// TwinCAT 3 PLC project PLC01
// ProgramVersion: 3.1.4024.0
// libraries:
//   Tc2_EtherCAT, * (Beckhoff Automation GmbH)
//   Tc2_Standard, * (Beckhoff Automation GmbH)
//   Tc2_System, * (Beckhoff Automation GmbH)
//   Tc2_Utilities, * (Beckhoff Automation GmbH)
//   Tc3_Module, * (Beckhoff Automation GmbH)
// project tree:
//   / GlobalTextList.TcGTLO, PlcTask.TcTTO, Visualization Manager.TcVMO (not stored)
//   GVLs/ G_Safety.TcGVL
//   POUs/ FB_Sample.TcPOU, FB_Teste.TcPOU, MAIN.TcPOU, safetyDiag.TcPOU
//   POUs/SafetyDiag/DUTs/ E_connInfoDiag.TcDUT, st_ConnectionInfoData.TcDUT, st_diagFBBits.TcDUT, st_infoDataFB.TcDUT, st_InfoDataGroup.TcDUT
//   POUs/SafetyDiag/ FB_ConnDiagELx904.TcPOU, FB_ConnectionDiag.TcPOU, FB_EStopDiag.TcPOU, FB_GroupDiag.TcPOU
//   POUs/SafetyDiag/ITF/ I_FBDiag.TcIO
//   VISUs/ ConnDiag.TcVIS, FB_Diag.TcVIS, footer.TcVIS, Group.TcVIS, Visualization.TcVIS
//   VISUs/Frames/ DiagConnELx904.TcVIS, DiagEStop.TcVIS
// real-time tasks:
//   TASK PlcTask: cycle T#10ms, priority 20, ADS port 350
// motion (NC):
//   TASK NC-Task 1 SAF: cycle T#2ms, priority 4, ADS port 501
//   TASK NC-Task 1 SVB: cycle T#10ms, priority 8, ADS port 511
//   AXIS Axis 1 (id 1)
//     OtherSettings: AllowMotionCmdToSlave=true
//     encoder EncType=19
//       EncPara: MaxCount=#xffffffff
//     drive DrvType=16
//       DrvPara: MaxCount=#xffffffff, DriveControlDWord=#x00020000
//         Analog: TorqueSetpointScale=10, ScaleFactorActTorque=0.1
//         TimeComp: TaskDelayCycles=1
//     controller CtrType=1
//       CtrPara: PriorControlFactor=1
//         Observer: BandWidth=20
//   AXIS Axis 2 (id 2)
//     OtherSettings: AllowMotionCmdToSlave=true
//     encoder EncType=19
//       EncPara: MaxCount=#xffffffff
//     drive DrvType=16
//       DrvPara: MaxCount=#xffffffff, DriveControlDWord=#x00020000
//         Analog: TorqueSetpointScale=10, ScaleFactorActTorque=0.1
//         TimeComp: TaskDelayCycles=1
//     controller CtrType=1
//       CtrPara: PriorControlFactor=1
//         Observer: BandWidth=20
// I/O:
//   DEVICE Device 2 (EtherCAT), AmsNetId 192.168.10.7.3.1
//     Term 1 (EK1100) [EK1100 EtherCAT Coupler (2A E-Bus)]
//       Term 2 (EL1012) [EL1012 2Ch. Dig. Input 24V, 10µs]
//       Term 3 (EL1012) [EL1012 2Ch. Dig. Input 24V, 10µs]
//       Term 4 (EL1012) [EL1012 2Ch. Dig. Input 24V, 10µs]
//       Term 5 (EL1012) [EL1012 2Ch. Dig. Input 24V, 10µs]
//       Term 6 (EL2004) [EL2004 4Ch. Dig. Output 24V, 0.5A]
//       Term 7 (EL4002) [EL4002 2Ch. Ana. Output 0-10V, 12bit]
//       Term 8 (EL9512) [EL9512 Power supply terminal 12V]
//       Term 9 (EL3102) [EL3102 2Ch. Ana. Input +/-10V, Diff.]
//       Term 16 (EL9011) [EL9011 End Terminal]
//     Term 10 (EK1100) [EK1100 EtherCAT Coupler (2A E-Bus)]
//       Term 11 (EL7211-0010) [EL7211-0010 1Ch. MDP742 Servo motor output stage with OCT (50V, 4.5A RMS)]
//       Term 12 (EL7211-0010) [EL7211-0010 1Ch. MDP742 Servo motor output stage with OCT (50V, 4.5A RMS)]
//       Term 13 (EL1904) [EL1904, 4 Ch. Safety Input 24V, TwinSAFE]
//         modules: Module 1 (FSOES)
//       Term 14 (EL2904) [EL2904, 4 Ch. Safety Output 24V, 0.5A, TwinSAFE]
//         modules: Module 1 (FSOES), Module 2 (DO)
//       Term 15 (EL6900) [EL6900, TwinSAFE PLC]
//       Term 17 (EL9011) [EL9011 End Terminal]
// variable links:
//   Device 2 (EtherCAT) <-> Device 2 (EtherCAT)/Term 10 (EK1100)/Term 13 (EL1904)
//     Term 10 (EK1100)/Term 15 (EL6900)/ConnectionInputs/Message_2 TxPDO <-> Module 1 (FSOES)/RxPDO/FSOE
//   Device 2 (EtherCAT) <-> Device 2 (EtherCAT)/Term 10 (EK1100)/Term 14 (EL2904)
//     Term 10 (EK1100)/Term 15 (EL6900)/ConnectionOutputs/Message_3 RxPDO <-> Module 1 (FSOES)/TxPDO/FSOE
//   Device 2 (EtherCAT) <-> Device 2 (EtherCAT)/Term 10 (EK1100)/Term 15 (EL6900)
//     Term 10 (EK1100)/Term 13 (EL1904)/Module 1 (FSOES)/TxPDO/FSOE <-> ConnectionOutputs/Message_2 RxPDO
//     Term 10 (EK1100)/Term 14 (EL2904)/Module 1 (FSOES)/RxPDO/FSOE <-> ConnectionInputs/Message_3 TxPDO
//   NC-Task 1 SAF/Axes/Axis 1 <-> Device 2 (EtherCAT)/Term 10 (EK1100)/Term 11 (EL7211-0010)
//     Drive/Inputs/In/nDcOutputTime <-> InfoData/DcOutputShift
//     Drive/Inputs/In/nState1 <-> DRV Statusword/Statusword
//     Drive/Inputs/In/nState2 <-> DRV Statusword/Statusword @bit 8
//     Drive/Inputs/In/nState4 @bit 1 <-> WcState/InputToggle
//     Drive/Inputs/In/nState4 <-> WcState/WcState
//     Drive/Outputs/Out/nCtrl1 <-> DRV Controlword/Controlword
//     Drive/Outputs/Out/nCtrl2 <-> DRV Controlword/Controlword @bit 8
//     Drive/Outputs/Out/nDataOut2 <-> DRV Target velocity/Target velocity
//     Enc/Inputs/In/nDataIn1 <-> FB Position/Position
//     Enc/Inputs/In/nDcInputTime <-> InfoData/DcInputShift
//     Enc/Inputs/In/nState4 @bit 1 <-> WcState/InputToggle
//     Enc/Inputs/In/nState4 <-> WcState/WcState
//   NC-Task 1 SAF/Axes/Axis 2 <-> Device 2 (EtherCAT)/Term 10 (EK1100)/Term 12 (EL7211-0010)
//     Drive/Inputs/In/nDcOutputTime <-> InfoData/DcOutputShift
//     Drive/Inputs/In/nState1 <-> DRV Statusword/Statusword
//     Drive/Inputs/In/nState2 <-> DRV Statusword/Statusword @bit 8
//     Drive/Inputs/In/nState4 @bit 1 <-> WcState/InputToggle
//     Drive/Inputs/In/nState4 <-> WcState/WcState
//     Drive/Outputs/Out/nCtrl1 <-> DRV Controlword/Controlword
//     Drive/Outputs/Out/nCtrl2 <-> DRV Controlword/Controlword @bit 8
//     Drive/Outputs/Out/nDataOut2 <-> DRV Target velocity/Target velocity
//     Enc/Inputs/In/nDataIn1 <-> FB Position/Position
//     Enc/Inputs/In/nDcInputTime <-> InfoData/DcInputShift
//     Enc/Inputs/In/nState4 @bit 1 <-> WcState/InputToggle
//     Enc/Inputs/In/nState4 <-> WcState/WcState
//   PLC01/PLC01 Instance <-> Device 2 (EtherCAT)/Term 10 (EK1100)/Term 15 (EL6900)
//     PlcTask Inputs/safetyDiag.blocoEStop.fbInfoData/diag <-> Function Block Info Data/TwinSafeGroup1.Network1.FBEstop1 Info Data/Diag
//     PlcTask Inputs/safetyDiag.blocoEStop.fbInfoData/state <-> Function Block Info Data/TwinSafeGroup1.Network1.FBEstop1 Info Data/State
//     PlcTask Inputs/safetyDiag.connDiagEL1904.connInfo/bit{1..4} <-> Connection Info Data/Message_2 Info Data/Input Safe Data InputChannel{1..4}  (4 links)
//     PlcTask Inputs/safetyDiag.connDiagEL1904.connInfo/diag <-> Connection Info Data/Message_2 Info Data/Diag
//     PlcTask Inputs/safetyDiag.connDiagEL2904.connInfo/diag <-> Connection Info Data/Message_3 Info Data/Diag
//     PlcTask Inputs/safetyDiag.connDiagEL1904.connInfo/state <-> Connection Info Data/Message_2 Info Data/State
//     PlcTask Inputs/safetyDiag.connDiagEL2904.connInfo/state <-> Connection Info Data/Message_3 Info Data/State
//     PlcTask Inputs/safetyDiag.connDiagEL2904.connInfo/bit{1..4} <-> Connection Info Data/Message_3 Info Data/Output Safe Data OutputChannel{1..4}  (4 links)
//     PlcTask Inputs/safetyDiag.eStopGroup.groupInfoData <-> TwinSAFE Group Info Data/TwinSafeGroup1 Info Data
//     PlcTask Outputs/G_Safety.resetSafety <-> StandardOutputs/Standard In Var 1
//     PlcTask Outputs/G_Safety.runSafety <-> StandardOutputs/Standard In Var 4

CONFIGURATION PLC01
    RESOURCE PLC ON TwinCAT3
        TASK PlcTask(INTERVAL := T#10ms, PRIORITY := 20);
        PROGRAM MAIN WITH PlcTask : MAIN;
    END_RESOURCE
END_CONFIGURATION

// ---- POUs/SafetyDiag/DUTs/E_connInfoDiag.TcDUT
{attribute 'qualified_only'}
{attribute 'strict'}
TYPE E_connInfoDiag :
(
	invalidCommand,
	unknownCommand,
	invalidConnectionId,
	invalidCRC,
	watchdogTime,
	invalidFSOEAddr,
	invalidData,
	invalidCommParaLen,
	invalidCommPara,
	invalidUserParaLen,
	invalidUserPara,
	FSOEMasterReset,
	moduleErrOnSlave,
	moduleErrEl290x,
	slaveNotStarted,
	FSOESlaveErr,
	FSOESlaveFailsafeActive,
	startup,
	FSOEMasterFailsafeActive
);
END_TYPE

// ---- POUs/SafetyDiag/DUTs/st_ConnectionInfoData.TcDUT
TYPE st_ConnectionInfoData :
STRUCT
	state,diag:USINT;
	bit1,bit2,bit3,bit4:BIT;
END_STRUCT
END_TYPE

// ---- POUs/SafetyDiag/DUTs/st_diagFBBits.TcDUT
TYPE st_diagFBBits :ARRAY[0..15] OF BOOL;
END_TYPE

// ---- POUs/SafetyDiag/DUTs/st_infoDataFB.TcDUT
TYPE st_infoDataFB :
STRUCT
	state:USINT;
	diag:UINT;
END_STRUCT
END_TYPE

// ---- POUs/SafetyDiag/DUTs/st_InfoDataGroup.TcDUT
TYPE st_InfoDataGroup :
STRUCT
	state,diag:USINT;
END_STRUCT
END_TYPE

// ---- GVLs/G_Safety.TcGVL
{attribute 'qualified_only'}
VAR_GLOBAL
	runSafety AT %Q*:BOOL;	//ativação do safety
	resetSafety AT %Q*:BOOL;//reset do safety
END_VAR

// ---- POUs/SafetyDiag/ITF/I_FBDiag.TcIO
INTERFACE I_FBDiag

PROPERTY P_diagBits : st_diagFBBits
GET
END_GET
END_PROPERTY

PROPERTY P_State : STRING(20)
GET
END_GET
END_PROPERTY

END_INTERFACE

// ---- POUs/MAIN.TcPOU
PROGRAM MAIN
VAR
	r1:LREAL:=20;
    fbSample : FB_Sample; 
    sMyPath : STRING; 
	teste:FB_Teste;
	grupo:FB_GroupDiag;
END_VAR

safetyDiag();
fbSample(); 
sMyPath := fbSample.sPath;

END_PROGRAM

// ---- POUs/FB_Sample.TcPOU
{attribute 'reflection'} 
FUNCTION_BLOCK FB_Sample 
VAR 
    {attribute 'instance-path'} 
    {attribute 'noinit'} 
    sPath : STRING; 
END_VAR

END_FUNCTION_BLOCK

// ---- POUs/FB_Teste.TcPOU
{attribute 'reflection'} 
FUNCTION_BLOCK FB_Teste
VAR
    {attribute 'instance-path'} 
    {attribute 'noinit'} 
	varTeste:STRING;
END_VAR

END_FUNCTION_BLOCK

// ---- POUs/SafetyDiag/FB_GroupDiag.TcPOU
{attribute 'reflection'} 
FUNCTION_BLOCK FB_GroupDiag
VAR_INPUT
	logGroupErrorState:BOOL:=TRUE;
END_VAR
VAR
    {attribute 'instance-path'}
    {attribute 'noinit'}
	sPath:STRING;	
	groupInfoData AT %I*:st_InfoDataGroup;
	oldGroupState:USINT;
	sCurrDiag:STRING(20);
END_VAR

PROPERTY diagInfo : string(20)
GET
VAR
	s1:STRING(20);
END_VAR
CASE groupInfoData.diag OF
	0:s1:='';
	1:s1:='FBERROR';
	2:s1:='COMERROR';
	3:s1:='MODULEERROR';
	4:s1:='CMPERROR';
	5:s1:='DEACTIVATEERROR';
	6:s1:='RESTARTERROR';
END_CASE
diagInfo:=sCurrDiag:=s1;
END_GET
END_PROPERTY

METHOD PRIVATE M_GroupErrorLog : BOOL
VAR_INPUT
	groupName:STRING;
END_VAR
ADSLOGSTR(ADSLOG_MSGTYPE_ERROR OR ADSLOG_MSGTYPE_STRING,'Erro no grupo e diagnótico = %s' ,concat(groupName,concat(' , ',diagInfo)));
END_METHOD

PROPERTY stateInfo : string(20)
GET
VAR
	s1:STRING(20);
END_VAR
CASE groupInfoData.state OF
	1:s1:='RUN';
	2:s1:='STOP';
	4:s1:='ERROR';
		IF oldGroupState <> groupInfoData.state AND logGroupErrorState THEN
			M_GroupErrorLog(sPath);
		END_IF
	5:s1:='RESET';
	6:s1:='START';
	7:s1:='STOPERROR';
	16:s1:='DEACTIVATE';
	17:s1:='WAITCOMMERROR';
END_CASE
stateInfo:= s1;

oldGroupState:=groupInfoData.state;
END_GET
END_PROPERTY

END_FUNCTION_BLOCK

// ---- POUs/safetyDiag.TcPOU
PROGRAM safetyDiag
VAR
	fbDiag:I_FBDiag;
	blocoEStop:FB_EStopDiag;
	sEStopState: STRING(15);
	eStopDiagBits:st_diagFBBits;
	{region "Connection"}
	connDiagEL1904:FB_ConnDiagELx904;
	connDiagEL2904:FB_ConnDiagELx904;
	stateEL1904, stateEL2904:STRING(20);
	diagEL1904,diagEL2904:E_connInfoDiag;
	el1904Bits,el2904Bits:ARRAY[0..3] OF BOOL;
	{endregion}
	{region "GroupDiag"}
	eStopGroup:FB_GroupDiag;
	{endregion}
	groupState: STRING(20);
	sGroupDiagInfo: STRING(20);
END_VAR

fbDiag:=blocoEStop;
sEStopState:=fbDiag.P_State;
eStopDiagBits:=fbDiag.P_diagBits;


//Connection

stateEL1904:=connDiagEL1904.M_ConnInfoState();
stateEL2904:=connDiagEL2904.M_ConnInfoState();
diagEL1904:=connDiagEL1904.M_ConnInfoDiag();
diagEL2904:=connDiagEL2904.M_ConnInfoDiag();
el1904Bits:=connDiagEL1904.InputState;
el2904Bits:=connDiagEL2904.InputState;

//group
eStopGroup.logGroupErrorState:=TRUE;

groupState:=eStopGroup.stateInfo;
sGroupDiagInfo:=eStopGroup.diagInfo;

END_PROGRAM

// ---- POUs/SafetyDiag/FB_EStopDiag.TcPOU
FUNCTION_BLOCK FB_EStopDiag IMPLEMENTS I_FBDiag
VAR_INPUT
END_VAR
VAR_OUTPUT
END_VAR
VAR
	fbInfoData AT %I*:st_infoDataFB;
END_VAR

PROPERTY P_diagBits : st_diagFBBits
GET
VAR
	diagBits:st_diagFBBits;	
END_VAR
diagBits[0]:=fbInfoData.diag.0;
diagBits[1]:=fbInfoData.diag.1;
diagBits[2]:=fbInfoData.diag.2;
diagBits[3]:=fbInfoData.diag.3;
diagBits[4]:=fbInfoData.diag.4;
diagBits[5]:=fbInfoData.diag.5;
diagBits[6]:=fbInfoData.diag.6;
diagBits[7]:=fbInfoData.diag.7;
diagBits[8]:=fbInfoData.diag.8;
diagBits[9]:=fbInfoData.diag.9;
diagBits[10]:=fbInfoData.diag.10;
diagBits[11]:=fbInfoData.diag.11;
diagBits[12]:=fbInfoData.diag.12;
diagBits[13]:=fbInfoData.diag.13;
diagBits[14]:=fbInfoData.diag.14;
diagBits[15]:=fbInfoData.diag.15;

P_diagBits:= diagBits;
END_GET
END_PROPERTY

PROPERTY P_State : STRING(20)
GET
VAR
	state:STRING(20);
END_VAR
CASE fbInfoData.state OF
	0:state:='undefined';
	1:state:='RUN';
	2:state:='STOP';
	3:state:='SAFE';
	4:state:='ERROR';
	5:state:='RESET';
	6:state:='START';
	8:state:='DELAYOUT';
ELSE
	state:='Error';	
END_CASE
P_State:= state;
END_GET
END_PROPERTY

END_FUNCTION_BLOCK

// ---- POUs/SafetyDiag/FB_ConnDiagELx904.TcPOU
FUNCTION_BLOCK FB_ConnDiagELx904 EXTENDS FB_ConnectionDiag
VAR_INPUT
END_VAR
VAR_OUTPUT
END_VAR
VAR
END_VAR

PROPERTY InputState : ARRAY[0..3] OF BOOL
GET
VAR
	bits:ARRAY[0..3] OF BOOL;
END_VAR
bits[0]:= SUPER^.connInfo.bit1;
bits[1]:= SUPER^.connInfo.bit2;
bits[2]:= SUPER^.connInfo.bit3;
bits[3]:= SUPER^.connInfo.bit4;
InputState:=bits;
END_GET
END_PROPERTY

END_FUNCTION_BLOCK

// ---- POUs/SafetyDiag/FB_ConnectionDiag.TcPOU
FUNCTION_BLOCK FB_ConnectionDiag
VAR_INPUT
END_VAR
VAR_OUTPUT
END_VAR
VAR
	connInfo AT %I*:st_ConnectionInfoData;
END_VAR

METHOD M_ConnInfoDiag : E_connInfoDiag
VAR_INPUT
END_VAR
VAR 
	infoDiag:E_connInfoDiag;
END_VAR
CASE connInfo.diag OF
	1:infoDiag:=E_connInfoDiag.invalidCommand;
	2:infoDiag:=E_connInfoDiag.unknownCommand;
	3:infoDiag:=E_connInfoDiag.invalidConnectionId;
	4:infoDiag:=E_connInfoDiag.invalidCRC;
	5:infoDiag:=E_connInfoDiag.watchdogTime;
	6:infoDiag:=E_connInfoDiag.invalidFSOEAddr;
	7:infoDiag:=E_connInfoDiag.invalidData;
	8:infoDiag:=E_connInfoDiag.invalidCommParaLen;
	9:infoDiag:=E_connInfoDiag.invalidCommPara;
	10:infoDiag:=E_connInfoDiag.invalidUserParaLen;
	11:infoDiag:=E_connInfoDiag.invalidUserPara;
	12:infoDiag:=E_connInfoDiag.FSOEMasterReset;
	13:infoDiag:=E_connInfoDiag.moduleErrOnSlave;
	14:infoDiag:=E_connInfoDiag.moduleErrEl290x;
	15:infoDiag:=E_connInfoDiag.slaveNotStarted;
	16:infoDiag:=E_connInfoDiag.FSOESlaveErr;
	32:infoDiag:=E_connInfoDiag.FSOESlaveFailsafeActive;
	64:infoDiag:=E_connInfoDiag.startup;
	128:infoDiag:=E_connInfoDiag.FSOEMasterFailsafeActive;
END_CASE
M_ConnInfoDiag:=infoDiag;
END_METHOD

METHOD M_ConnInfoState : STRING(20)
VAR_INPUT
END_VAR
VAR
	s1:STRING(20);
END_VAR
CASE connInfo.state OF
	100:s1:='Reset State';
	101:s1:='Session State';
	102:s1:='Connection State';
	103:s1:='Parameter State';
	104:s1:='Data State';
	105:s1:='Shutdown State';
	106:s1:='Shutdown-Deactivate';
END_CASE
M_ConnInfoState:=s1;
END_METHOD

END_FUNCTION_BLOCK

// ---- GlobalTextList.TcGTLO
TEXTLIST GlobalTextList
  522 = '%s'
  254 = 'Conn Diag'
  105 = 'Diagnostic'
  934 = 'Discr. err grp 1, safe inputs'
  996 = 'Discr. err grp 2, safe inputs'
  875 = 'Discr. err grp 3, safe inputs'
  343 = 'Discr. err grp 4, safe inputs'
  562 = 'Discrepance err grp 1'
  683 = 'Discrepance err grp 1 '
  696 = 'Discrepance err grp 2'
  770 = 'Discrepance err grp 3'
  687 = 'Discrepance err grp 4'
  56 = 'FB diag'
  371 = 'Group Diag'
  314 = 'I/Os'
  195 = 'Label'
  856 = 'Monitoring err EDM 1'
  676 = 'Monitoring err EDM 2'
  641 = 'Reset'
  83 = 'Run'
  88 = 'State'
  586 = 'State: %s'
  809 = 'Tela 1'
END_TEXTLIST

// ---- VISUs/ConnDiag.TcVIS
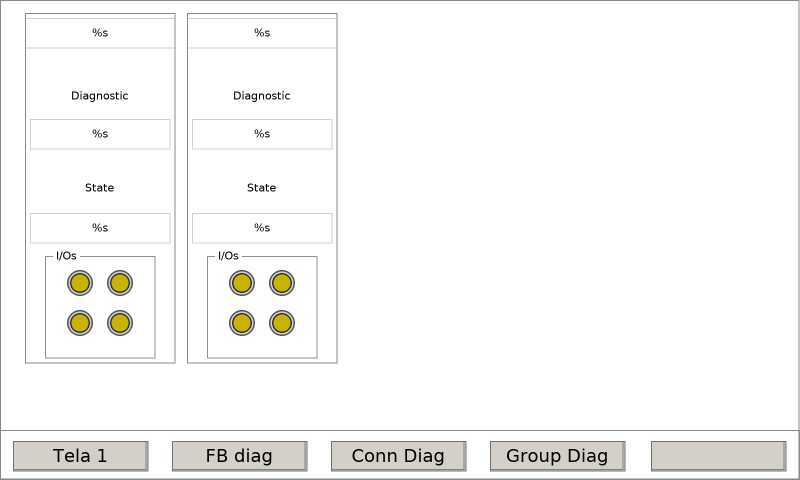
VISUALIZATION ConnDiag  // 800x480
    Frame (0,430 800x50)
        shows footer()
    Frame (25,13 150x350)
        shows DiagConnELx904(connName := 'EL 1904', diag := safetyDiag.diagEL1904, state := safetyDiag.stateEL1904, bits := safetyDiag.el1904Bits)
    Frame (187,13 150x350)
        shows DiagConnELx904(connName := 'EL 2904', diag := safetyDiag.diagEL2904, state := safetyDiag.stateEL2904, bits := safetyDiag.el2904Bits)
END_VISUALIZATION

// ---- VISUs/FB_Diag.TcVIS
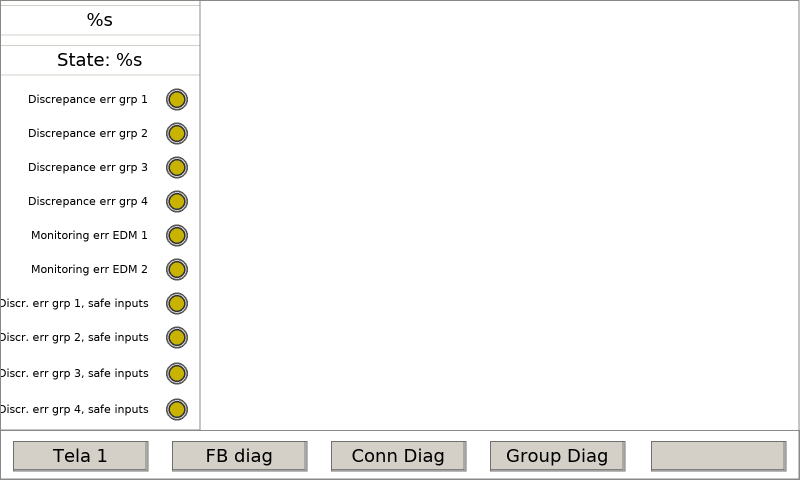
VISUALIZATION FB_Diag  // 800x480
    Frame (0,430 800x50)
        shows footer()
    Frame (0,0 200x430)
        shows DiagEStop(state := safetyDiag.sEStopState, bits := safetyDiag.eStopDiagBits, blockName := 'Emergência')
END_VISUALIZATION

// ---- VISUs/footer.TcVIS
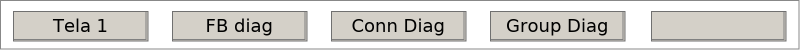
VISUALIZATION footer  // 800x50
    Button (13,11 135x30), "Tela 1"
        OnMouseClick: change screen: Visualization
    Button (172,11 135x30), "FB diag"
        OnMouseClick: change screen: FB_Diag
    Button (331,11 135x30), "Conn Diag"
        OnMouseClick: change screen: ConnDiag
    Button (490,11 135x30), "Group Diag"
        OnMouseClick: change screen: Group
    Button (651,11 135x30)
END_VISUALIZATION

// ---- VISUs/Frames/DiagConnELx904.TcVIS
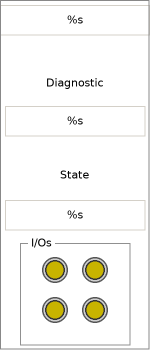
VISUALIZATION DiagConnELx904  // 150x350
VAR_INPUT
	connName:STRING(20);
	diag:E_connInfoDiag;
	state:STRING(20);
	bits:ARRAY[0..3] OF BOOL;
END_VAR
    GroupBox (20,235 110x110), "I/Os"
        Lamp1 (20,20 30x30), variable: bits[0], style: Lamp-Lamp1-Yellow
        Lamp1 (60,20 30x30), variable: bits[2], style: Lamp-Lamp1-Yellow
        Lamp1 (20,60 30x30), variable: bits[1], style: Lamp-Lamp1-Yellow
        Lamp1 (60,60 30x30), variable: bits[3], style: Lamp-Lamp1-Yellow
    Label (5,68 140x30), "Diagnostic"
    Label (5,160 140x30), "State"
    Textfield (5,106 140x30), "%s", text variable: diag
    Textfield (5,200 140x30), "%s", text variable: state
    Textfield (0,5 150x30), "%s", text variable: connName
END_VISUALIZATION

// ---- VISUs/Frames/DiagEStop.TcVIS
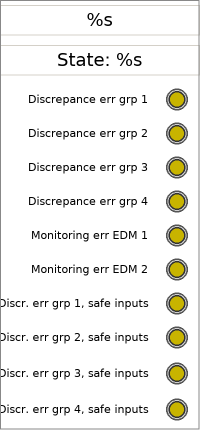
VISUALIZATION DiagEStop  // 200x430
VAR_INPUT
	state:STRING(15);
	bits:st_diagFBBits;
	blockName:STRING(15);
END_VAR
    Label (1,87 150x25), "Discrepance err grp 1"
    Label (1,121 150x25), "Discrepance err grp 2"
    Label (1,155 150x25), "Discrepance err grp 3"
    Label (1,189 150x25), "Discrepance err grp 4"
    Label (1,223 150x25), "Monitoring err EDM 1"
    Label (1,257 150x25), "Monitoring err EDM 2"
    Label (1,291 150x25), "Discr. err grp 1, safe inputs"
    Label (1,325 150x25), "Discr. err grp 2, safe inputs"
    Lamp1 (162,87 30x25), variable: bits[0], style: Lamp-Lamp1-Yellow
    Lamp1 (162,121 30x25), variable: bits[1], style: Lamp-Lamp1-Yellow
    Lamp1 (162,189 30x25), variable: bits[3], style: Lamp-Lamp1-Yellow
    Lamp1 (162,223 30x25), variable: bits[4], style: Lamp-Lamp1-Yellow
    Lamp1 (162,257 30x25), variable: bits[5], style: Lamp-Lamp1-Yellow
    Lamp1 (162,291 30x25), variable: bits[8], style: Lamp-Lamp1-Yellow
    Lamp1 (162,325 30x25), variable: bits[9], style: Lamp-Lamp1-Yellow
    Lamp1 (162,155 30x25), variable: bits[2], style: Lamp-Lamp1-Yellow
    Label (1,361 150x25), "Discr. err grp 3, safe inputs"
    Lamp1 (162,361 30x25), variable: bits[10], style: Lamp-Lamp1-Yellow
    Label (1,397 150x25), "Discr. err grp 4, safe inputs"
    Lamp1 (162,397 30x25), variable: bits[11], style: Lamp-Lamp1-Yellow
    Textfield (0,45 200x30), "State: %s", text variable: state
    Textfield (0,5 200x30), "%s", text variable: blockName
END_VISUALIZATION

// ---- VISUs/Group.TcVIS
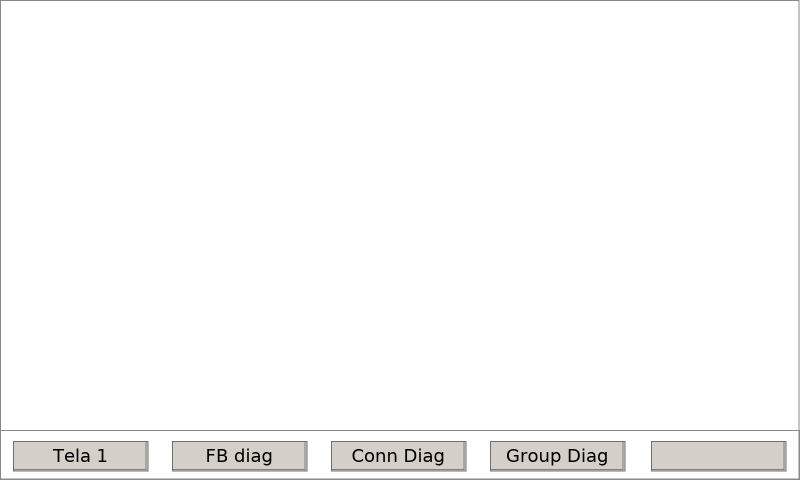
VISUALIZATION Group  // 800x480
    Frame (0,430 800x50)
        shows footer()
END_VISUALIZATION

// ---- VISUs/Visualization.TcVIS
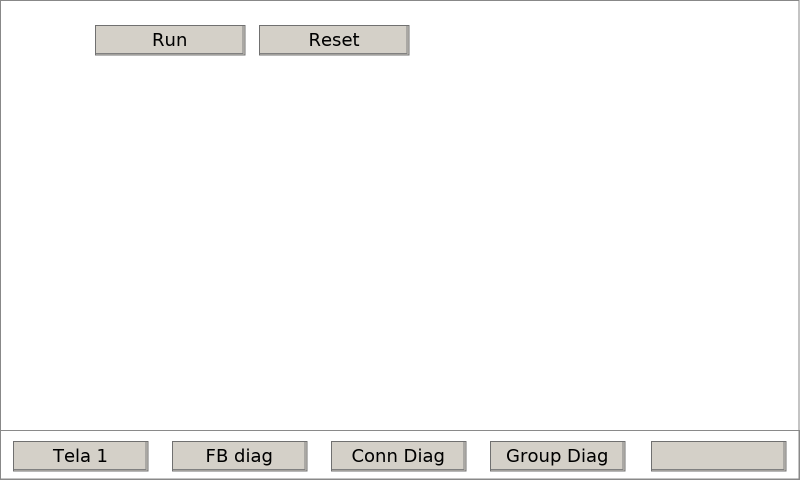
VISUALIZATION Visualization  // 800x480
    Button (95,25 150x30), "Run"
        toggle G_Safety.runSafety
    Button (259,25 150x30), "Reset"
        tap G_Safety.resetSafety
    Frame (0,430 800x50)
        shows footer()
END_VISUALIZATION
